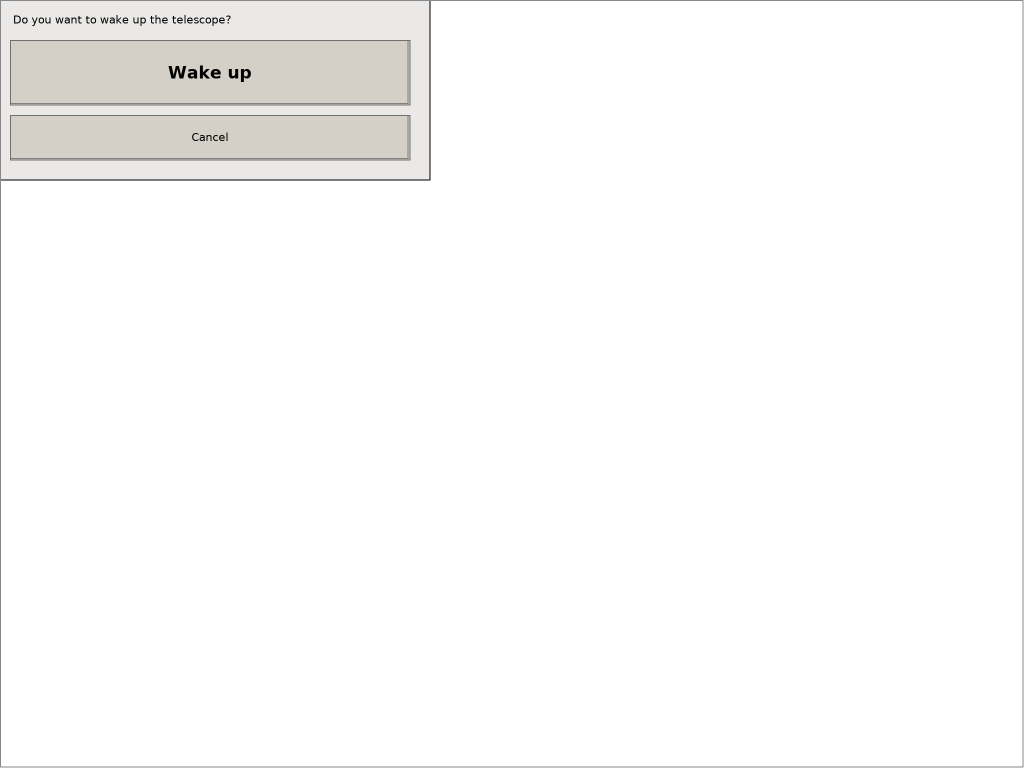
VISUALIZATION VISU_MTCSWakeUpTelescopeDialog  // 1024x768
    Rectangle (0,0 430x180)
    Button (10,40 400x65), "Wake up", input disabled if: GLOBAL.mtcs.processes.wakeUp.statuses.enabledStatus.disabled
        OnMouseClick: execute { GLOBAL.mtcs.processes.wakeUp.do_request := TRUE; }
        OnMouseClick: CloseDialog Dialog=VISU_MTCSWakeUpTelescopeDialog, Result=OK, NumpadKeypadSet=True
    Button (10,115 400x45), "Cancel"
        OnMouseClick: CloseDialog Dialog=VISU_MTCSWakeUpTelescopeDialog, Result=OK, NumpadKeypadSet=True
    Label (10,5 400x30), "Do you want to wake up the telescope?"
END_VISUALIZATION

(* stored: Version 1.1.0.1, ProductVersion 3.1.4018.5
   Visu VISU_MTCSWakeUpTelescopeDialog: Id {1c4ada83-f2a6-4bbe-add8-f035f1ce9849} *)
